Staubli VAL3: lists_string_num.pjx

--- lists_string_num.pjx ---
Parameters version=s8.13.1Cs9_BS2800 stackSize=5000 millimeterUnit=true
Data file=lists_string_num.dtx

--- lists_string_num.dtx ---
mdesc mNomSpeed
public string sString
public num nNum
